(* Logix 5000 project; controller RG_Chopper vendor 1 type 14 code 235 rev 32.12; software revision 32.04; part 3 of 6 *)
(* tags used below, declared in another part *)
   _ILG101_GREEN_PB : BOOL;   // Green Light Pushbutton Local:1:O.Data.2
   ALARM_FATAL : BOOL;   // Fatal Alarm Stops All Operation
   ALARM_GATE_OPEN : BOOL;   // Gate Open
   ALARM_LIGHT_CUR : BOOL;   // Light Curtain Obstructed
   ALARM_NON_FATAL : BOOL;
   BLANK_LVL_DISP : BOOL;   // Disables Tank Level Display
   CIP_CAUSTIC_RUNNING : ALIAS FOR SIGNAL_OUT_RG_CHOPPER.4;
   CIP_CMPLT : BOOL;   // CIP Complete Indicator
   CIP_COMPLETE : ALIAS FOR SIGNAL_IN_RG_CHOPPER.4;
   CIP_CYC_ST : DINT;   // CIP Cycle Status HMI
   CIP_OUT : DINT;   // CIP Output Bits
   CIP_STEP : COUNTER;   // CIP Step Counter
   CIP_STEP_BIT : DINT;   // CIP Step Enable Bit
   CIP_STEP_DN : BOOL;   // CIP Step Done
   CIP_STEP_TMR : TIMER;   // CIP Step Timer
   CIP_STP_TM_TB : DINT[13];   // CIP Step Timer PreSet Table
   CIP_STRT_RUN : BOOL;   // CIP System Started
   CIP_WATER_RUNNING : ALIAS FOR SIGNAL_OUT_RG_CHOPPER.3;
   CYC_CIP : BOOL;   // CIP Cycle Running
   CYC_RUN : BOOL;   // Production Cycle Running
   CYC_ST : DINT;
   DBX101_AM : PUSH_PUSH_PB;   // DBX-101 Push-Push Button Control
   DBX101_AUX : BOOL;   // DBX-101 Agitator Motor Aux
   DBX101_CTL : HOA_CTRL_v2;   // DBX-101 Agitator Motor Control Block
   DBX101_CTL_ST : DINT;   // DBX-101 Control Status 0= Auto 1= Manual 2= Error
   DBX101_FAULT : BOOL;
   DBX101_MAN : PUSH_PUSH_PB;   // DBX-101 Manual Run Push-Push
   DBX101_MAN_RUN : BOOL;   // DBX-101 Manual Run
   DBX101_MAN_ST : DINT;   // DBX-101 Manual Control Status
   DBX101_PB : BOOL;   // DBX-101 Auto / Manual Push-Push Button
   DBX101_STS : DINT;   // DBX-101 Agitator Motor Status (HMI)
   DBX102_AM : PUSH_PUSH_PB;   // DBX-102 Push-Push Button Control
   DBX102_AUX : ALIAS FOR SIGNAL_IN_RG_CHOPPER.0;   // DBX-102 VFD Active AUX
   DBX102_CTL : HOA_CTRL_v2;   // DBX102 Product Discharge Pump Control Block
   DBX102_CTL_ST : DINT;   // DBX-102 Control Status 0= Auto 1= Manual 2= Error
   DBX102_M_FAULT : BOOL;   // DBX-102 Discharge Pump Drive or Motor Fault
   DBX102_MAN : PUSH_PUSH_PB;   // DBX-102 Manual Control Push-Push
   DBX102_MAN_RUN : BOOL;   // DBX-102 Manual Mode Run PB
   DBX102_MAN_ST : DINT;   // DBX-102 Manual Control Status
   DBX102_PB : BOOL;   // DBX-102 Auto / Manual Push-Push Button
   DBX102_SPD_AM : PUSH_PUSH_PB;   // DBX-102 Speed Push-Push Button Control
   DBX102_SPD_ST : DINT;   // DBX-102 VFD Speed Control Status 0= Auto 1= Manual 2= Error
   DBX102_STS : DINT;   // DBX-102 Product Pump Status (HMI)
   DBX102_VFD_FB : ANLG_SCALE;   // DBX-102 VFD Speed FB Scaling (HMI)
   DBX102_VFD_FB_SCL : REAL;   // DBX-102 Product Pump VFD Speed FB Scaling (HMI)
   DBX103_AM : PUSH_PUSH_PB;   // DBX-103 Push-Push Button Control
   DBX103_AUX : BOOL;   // DBX-103 Water Pump Aux
   DBX103_CTL : HOA_CTRL_v2;   // DBX-103 Hot Water Pump Control Block
   DBX103_CTL_ST : DINT;   // DBX-103 Control Status 1= Auto 2= Manual 3= Error
   DBX103_FAULT : BOOL;   // DBX-103 Hot Water Pump Fault
   DBX103_MAN : PUSH_PUSH_PB;   // DBX-103 Manual Run Push-Push
   DBX103_MAN_RUN : BOOL;   // DBX-101 Manual Run
   DBX103_MAN_ST : DINT;   // DBX-103 Manual Control Status
   DBX103_PB : BOOL;   // DBX-103 Auto / Manual Push-Push Button
   DBX103_STS : DINT;   // DBX-103 Hot Water Pump Status (HMI)
   DBX104_AM : PUSH_PUSH_PB;   // DBX-104 Push-Push Button Control
   DBX104_AUX : BOOL;   // DBX-104 VFD Active AUX
   DBX104_CTL : HOA_CTRL_v2;   // DBX-104 Reversing Motor Starter Control
   DBX104_CTL_ST : DINT;   // DBX-104 Control Status 0= Auto 1= Manual 2= Error
   DBX104_FAULT : BOOL;   // DBX-104 Dumper Elevator Drive Fault
   DBX104_M_FAULT : BOOL;   // DBX-104 Dumper Elevator Drive or Motor Fault
   DBX104_MAN : PUSH_PUSH_PB;   // DBX-104 Manual Control Push-Push
   DBX104_MAN_RUN : BOOL;   // DBX-104 Manual Mode Run PB
   DBX104_MAN_ST : DINT;   // DBX-104 Manual Control Status
   DBX104_PB : BOOL;   // DBX-104 Auto / Manual Push-Push Button
   DBX104_SPD_AM : PUSH_PUSH_PB;   // DBX-104 Speed Push-Push Button Control
   DBX104_SPD_ST : DINT;   // DBX-104 VFD Speed Control Status 0= Auto 1= Manual 2= Error
   DBX104_STS : DINT;   // DBX-104 Product Pump Status (HMI)
   DBX104_VFD_FB : ANLG_SCALE;   // DBX-104 VFD Speed FB Scaling (HMI)
   DBX104_VFD_FB_SCL : REAL;   // DBX-104 Product Pump VFD Speed FB Scaling (HMI)
   DL101_Scl : REAL;
   DTT102 : REAL;   // Discharge Product Temperature
   DWN_MKBK : BOOL;   // Elevator Down Make / Break LS_L1 Detection
   DWN_OT_AL : BOOL;   // New Dumper DOWN Over Travel Alarm
   Fault_ACK : BOOL;   // Fault Acknowledge
   Flash : BOOL;
   Gate_SW1 : DCI_MONITOR;   // Safety Switch Gate_SW1 SW105 A/B
   Gate_SW2 : DCI_MONITOR;   // Safety Switch Gate_SW2 SW108 A/B
   HI_PROD_TEMP_AL : BOOL;   // Product Temperature High Alarm
   HI_PROD_TEMP_SP : REAL;   // Product High Temperature Alarm SetPoint
   HI_TMP_TMR : TIMER;   // Product Temperature High Alarm Timer
   HMI_USER : STRING;   // Current Logged HMI User
   ILG104_GREEN_STACK : BOOL;   // Stack Light Green
   ILG105_YELLOW_STACK : BOOL;   // Stack Light Yellow
   ILG106_RED_STACK : BOOL;   // Stack Light Red
   L_CRASH_ALM : BOOL;   // New Dumper Lower CRASH Alarm
   LSS_LOT1 : BOOL;   // New Dumper LOWER OVER TRAVEL Limit Switch
   LVL_BLANK_SP : REAL;   // Real Value Below Blanks Level Display
   LVL_LO_TMR : TIMER;   // Low Tank Level Alarm Debounce Timer
   M104S_DWN_CTL : CONFIGURABLE_ROUT;   // DBX-104 Dump Elevator Safety Starter Down Output
   M104S_STRT_CTL : CONFIGURABLE_ROUT;   // DBX-104 Dump Elevator Safety Starter Enable Output
   M104S_UP_CTL : CONFIGURABLE_ROUT;   // DBX-104 Dump Elevator Safety Starter UP Output
   NO_USER : BOOL;   // No HMI User Logged on
   ONESHOT : DINT;   // One-shot Word
   PROC_TMR : TIMER[16];   // Process Timers
   S_ESTOP : BOOL;   // Safety ESTOP
   SHTDWN_ACTV : BOOL;   // System Shutdown is In Progress
   SHTDWN_CMPLT : BOOL;   // System Shutdown Complete
   SHUTDOWN : DINT;   // System Shutdown Control Bits
   SIGNAL_OUT_RG_CHOPPER : DINT;
   START_CMPLT : BOOL;   // System Start up Complete
   SW102_STOP_PB : BOOL;   // Stop PB HMI
   SW103_CIP_PB : BOOL;   // CIP PB HMI
   SW104_ESTOP : BOOL;   // Safety E-Stop SW-104
   SW106_LC : LIGHT_CURTAIN;   // Safety SW106 Light Curain
   SW107_TANK_LID : BOOL;   // Tank Lid Safety Switch Active
   SYS_OK : BOOL;   // System OK No Fatal Alarms
   SYS_STRT_RUN : BOOL;   // System Start / Run
   TCV101_CTL : PID;   // PCV-101 PID Temperature Control
   UP_MKBK : BOOL;   // Elevator Down Make / Break LS_U1 Detection
   UP_OT_AL : BOOL;   // New Dumper UP Over Travel Alarm
   USER_ON : BOOL;   // There IS a valid HMI User Logged On
   WTR_HI_TEMP : BOOL;   // High Water Temperature Alarm
   WTR_HI_TMR : TIMER;   // High Water Temperature Alarm Debounce Timer

PROGRAM MainProgram   (* main routine MainRoutine *)
VAR
   L2_FAIL_TMR : TIMER := (PRE := 4000);   // LSSL2 Fail Always Open Detect
   LSSL2_FAIL : BOOL;   // Lower Safety Limit Switch LSS-L2 Fail
   LSSL2_FAIL2 : BOOL;   // Lower Safety Limit Switch LSS-L2 Mode 2
   LSSU2_FAIL : BOOL;   // Upper Safety Limit Switch LSS-U2 Fail
   LSSU2_FAIL2 : BOOL;   // Upper Safety Limit Switch USS-L2 Mode 2
   U2_FAIL_TMR : TIMER := (PRE := 4000);   // LSSU2 Fail Always Open Detect
END_VAR

ROUTINE ALARMS   (* ladder *)
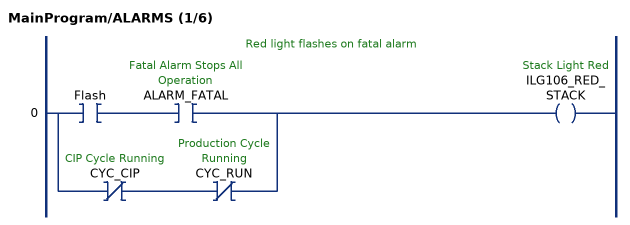
   // Red light flashes on fatal alarm
   0: [XIC(Flash) XIC(ALARM_FATAL) ,XIO(CYC_CIP) XIO(CYC_RUN) ]OTE(ILG106_RED_STACK);
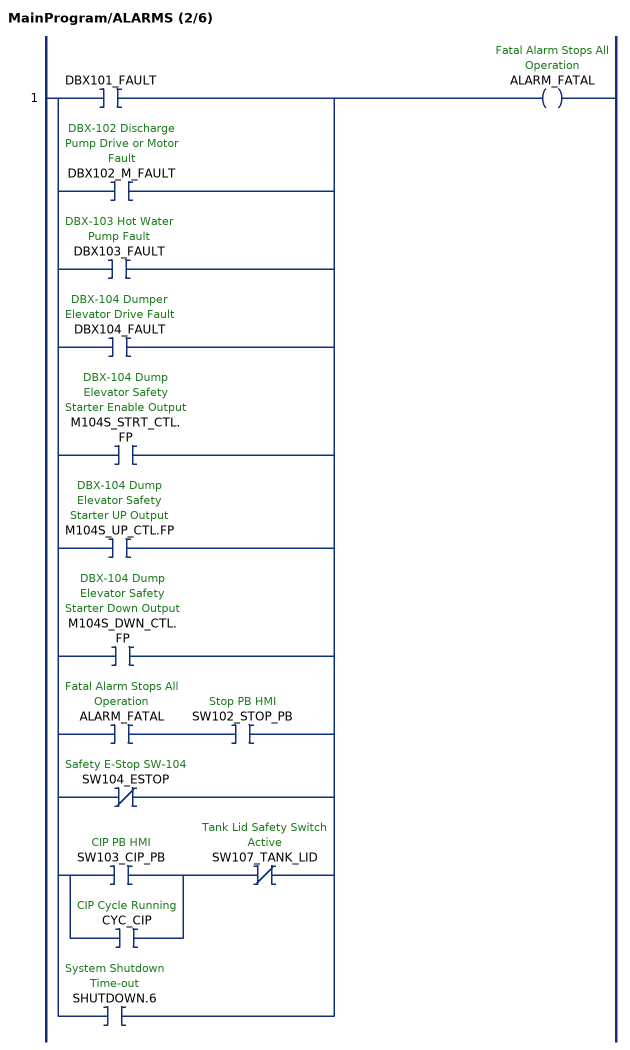
   1: [XIC(DBX101_FAULT) ,XIC(DBX102_M_FAULT) ,XIC(DBX103_FAULT) ,XIC(DBX104_FAULT) ,XIC(M104S_STRT_CTL.FP) ,XIC(M104S_UP_CTL.FP) ,XIC(M104S_DWN_CTL.FP) ,XIC(ALARM_FATAL) XIC(SW102_STOP_PB) ,XIO(SW104_ESTOP) ,[XIC(SW103_CIP_PB) ,XIC(CYC_CIP) ] XIO(SW107_TANK_LID) ,XIC(SHUTDOWN.6) ]OTE(ALARM_FATAL);
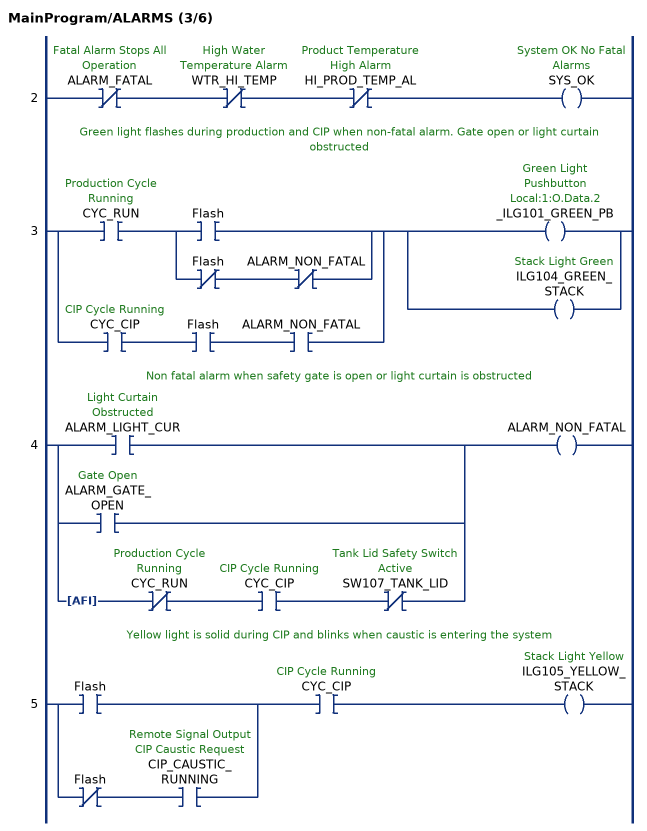
   2: XIO(ALARM_FATAL)XIO(WTR_HI_TEMP)XIO(HI_PROD_TEMP_AL)OTE(SYS_OK);
   // Green light flashes during production and CIP when non-fatal alarm. Gate open or light curtain obstructed
   3: [XIC(CYC_RUN) [XIC(Flash) ,XIO(Flash) XIO(ALARM_NON_FATAL) ] ,XIC(CYC_CIP) XIC(Flash) XIC(ALARM_NON_FATAL) ][OTE(_ILG101_GREEN_PB) ,OTE(ILG104_GREEN_STACK) ];
   // Non fatal alarm when safety gate is open or light curtain is obstructed
   4: [XIC(ALARM_LIGHT_CUR) ,XIC(ALARM_GATE_OPEN) ,AFI() XIO(CYC_RUN) XIC(CYC_CIP) XIO(SW107_TANK_LID) ]OTE(ALARM_NON_FATAL);
   // Yellow light is solid during CIP and blinks when caustic is entering the system
   5: [XIC(Flash) ,XIO(Flash) XIC(CIP_CAUSTIC_RUNNING) ]XIC(CYC_CIP)OTE(ILG105_YELLOW_STACK);
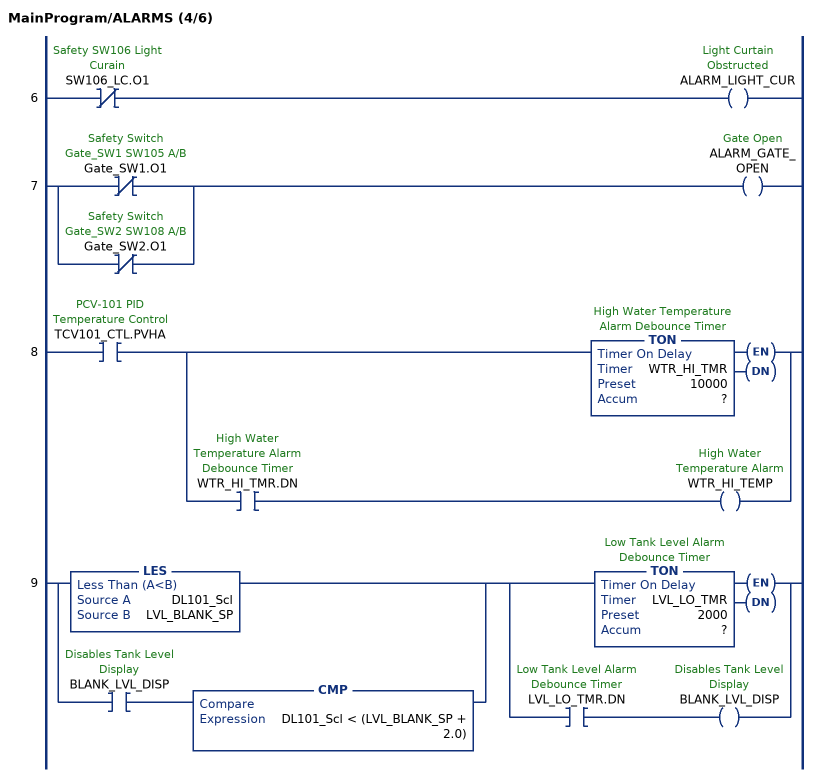
   6: XIO(SW106_LC.O1)OTE(ALARM_LIGHT_CUR);
   7: [XIO(Gate_SW1.O1) ,XIO(Gate_SW2.O1) ]OTE(ALARM_GATE_OPEN);
   8: XIC(TCV101_CTL.PVHA)[TON(WTR_HI_TMR,?,?) ,XIC(WTR_HI_TMR.DN) OTE(WTR_HI_TEMP) ];
   9: [LES(DL101_Scl,LVL_BLANK_SP) ,XIC(BLANK_LVL_DISP) CMP(DL101_Scl < (LVL_BLANK_SP + 2.0)) ][TON(LVL_LO_TMR,?,?) ,XIC(LVL_LO_TMR.DN) OTE(BLANK_LVL_DISP) ];
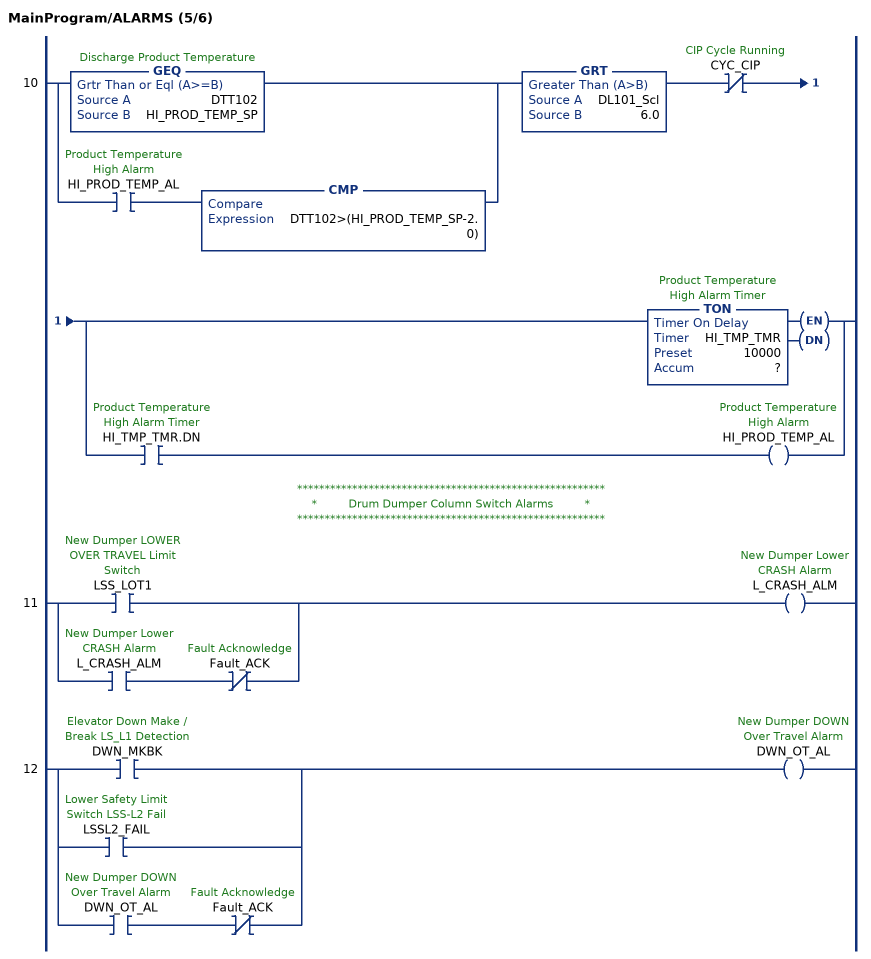
   10: [GEQ(DTT102,HI_PROD_TEMP_SP) ,XIC(HI_PROD_TEMP_AL) CMP(DTT102>(HI_PROD_TEMP_SP-2.0)) ]GRT(DL101_Scl,6.0)XIO(CYC_CIP)[TON(HI_TMP_TMR,?,?) ,XIC(HI_TMP_TMR.DN) OTE(HI_PROD_TEMP_AL) ];
   // ********************************************************
   // *         Drum Dumper Column Switch Alarms         *
   // ********************************************************
   11: [XIC(LSS_LOT1) ,XIC(L_CRASH_ALM) XIO(Fault_ACK) ]OTE(L_CRASH_ALM);
   12: [XIC(DWN_MKBK) ,XIC(LSSL2_FAIL) ,XIC(DWN_OT_AL) XIO(Fault_ACK) ]OTE(DWN_OT_AL);
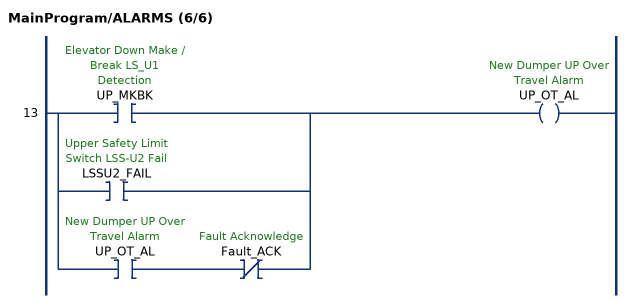
   13: [XIC(UP_MKBK) ,XIC(LSSU2_FAIL) ,XIC(UP_OT_AL) XIO(Fault_ACK) ]OTE(UP_OT_AL);
END_ROUTINE

ROUTINE CIP   (* ladder *)
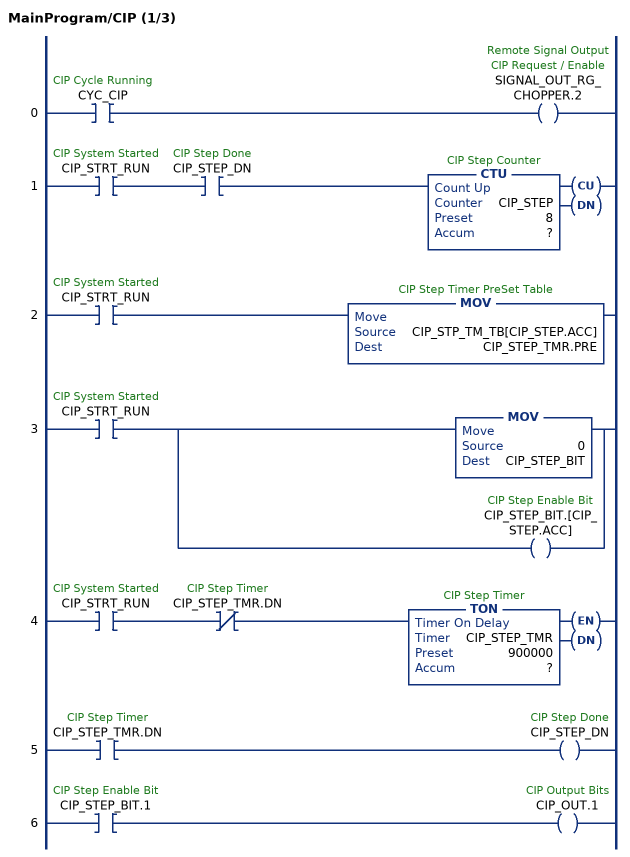
   0: XIC(CYC_CIP)OTE(SIGNAL_OUT_RG_CHOPPER.2);
   1: XIC(CIP_STRT_RUN)XIC(CIP_STEP_DN)CTU(CIP_STEP,?,?);
   2: XIC(CIP_STRT_RUN)MOV(CIP_STP_TM_TB[CIP_STEP.ACC],CIP_STEP_TMR.PRE);
   3: XIC(CIP_STRT_RUN)[MOV(0,CIP_STEP_BIT) ,OTE(CIP_STEP_BIT.[CIP_STEP.ACC]) ];
   4: XIC(CIP_STRT_RUN)XIO(CIP_STEP_TMR.DN)TON(CIP_STEP_TMR,?,?);
   5: XIC(CIP_STEP_TMR.DN)OTE(CIP_STEP_DN);
   6: XIC(CIP_STEP_BIT.1)OTE(CIP_OUT.1);
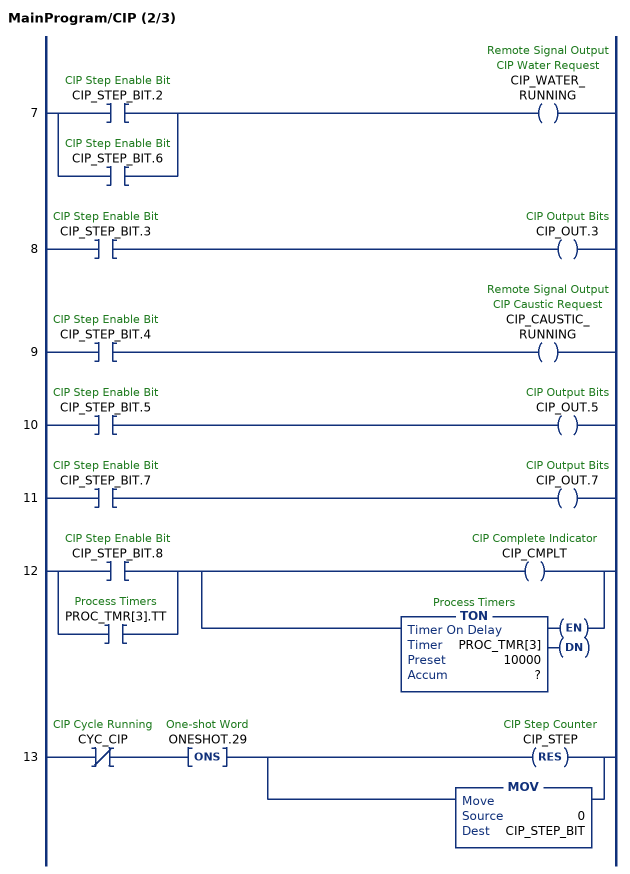
   7: [XIC(CIP_STEP_BIT.2) ,XIC(CIP_STEP_BIT.6) ]OTE(CIP_WATER_RUNNING);
   8: XIC(CIP_STEP_BIT.3)OTE(CIP_OUT.3);
   9: XIC(CIP_STEP_BIT.4)OTE(CIP_CAUSTIC_RUNNING);
   10: XIC(CIP_STEP_BIT.5)OTE(CIP_OUT.5);
   11: XIC(CIP_STEP_BIT.7)OTE(CIP_OUT.7);
   12: [XIC(CIP_STEP_BIT.8) ,XIC(PROC_TMR[3].TT) ][OTE(CIP_CMPLT) ,TON(PROC_TMR[3],?,?) ];
   13: XIO(CYC_CIP)ONS(ONESHOT.29)[RES(CIP_STEP) ,MOV(0,CIP_STEP_BIT) ];
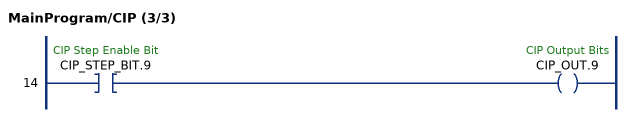
   14: XIC(CIP_STEP_BIT.9)OTE(CIP_OUT.9);
END_ROUTINE

ROUTINE HMI   (* ladder *)
// HMI Interface Code
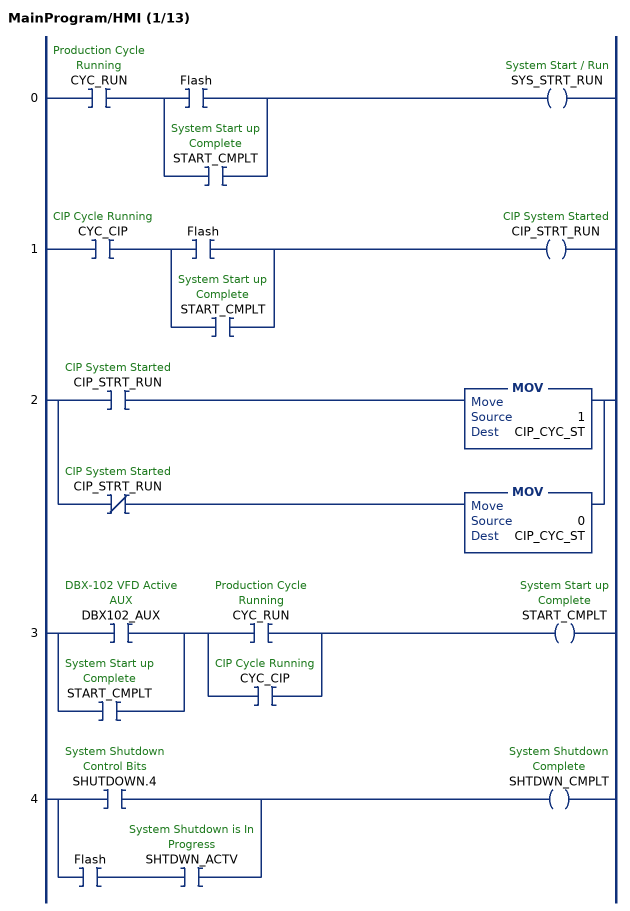
   0: XIC(CYC_RUN)[XIC(Flash) ,XIC(START_CMPLT) ]OTE(SYS_STRT_RUN);
   1: XIC(CYC_CIP)[XIC(Flash) ,XIC(START_CMPLT) ]OTE(CIP_STRT_RUN);
   2: [XIC(CIP_STRT_RUN) MOV(1,CIP_CYC_ST) ,XIO(CIP_STRT_RUN) MOV(0,CIP_CYC_ST) ];
   3: [XIC(DBX102_AUX) ,XIC(START_CMPLT) ][XIC(CYC_RUN) ,XIC(CYC_CIP) ]OTE(START_CMPLT);
   4: [XIC(SHUTDOWN.4) ,XIC(Flash) XIC(SHTDWN_ACTV) ]OTE(SHTDWN_CMPLT);
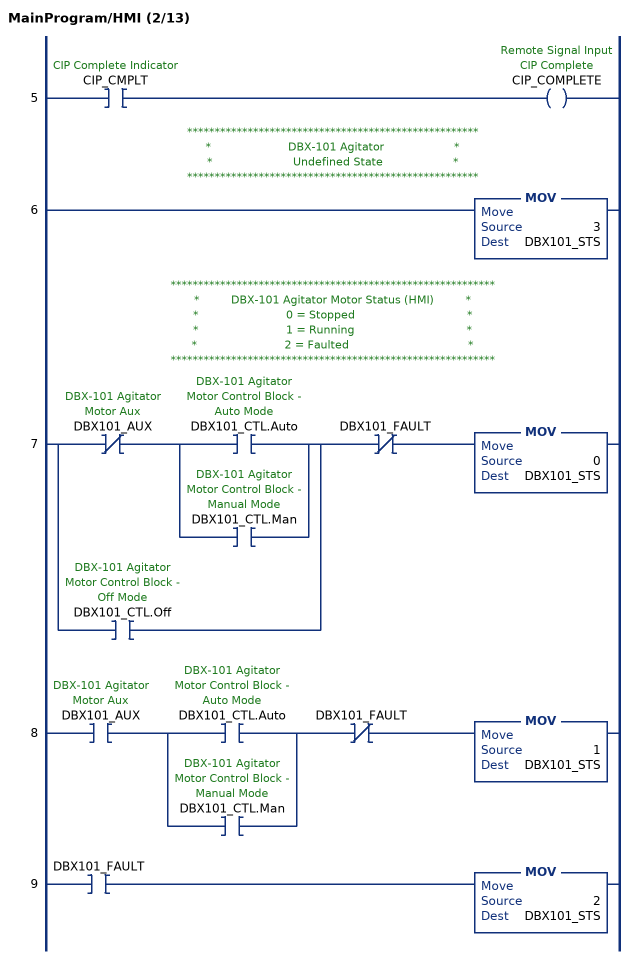
   5: XIC(CIP_CMPLT)OTE(CIP_COMPLETE);
   // *****************************************************
   // *                      DBX-101 Agitator                    *
   // *                       Undefined State                    *
   // *****************************************************
   6: MOV(3,DBX101_STS);
   // ***********************************************************
   // *         DBX-101 Agitator Motor Status (HMI)         *
   // *                         0 = Stopped                                *
   // *                         1 = Running                                *
   // *                         2 = Faulted                                  *
   // ***********************************************************
   7: [XIO(DBX101_AUX) [XIC(DBX101_CTL.Auto) ,XIC(DBX101_CTL.Man) ] ,XIC(DBX101_CTL.Off) ]XIO(DBX101_FAULT)MOV(0,DBX101_STS);
   8: XIC(DBX101_AUX)[XIC(DBX101_CTL.Auto) ,XIC(DBX101_CTL.Man) ]XIO(DBX101_FAULT)MOV(1,DBX101_STS);
   9: XIC(DBX101_FAULT)MOV(2,DBX101_STS);
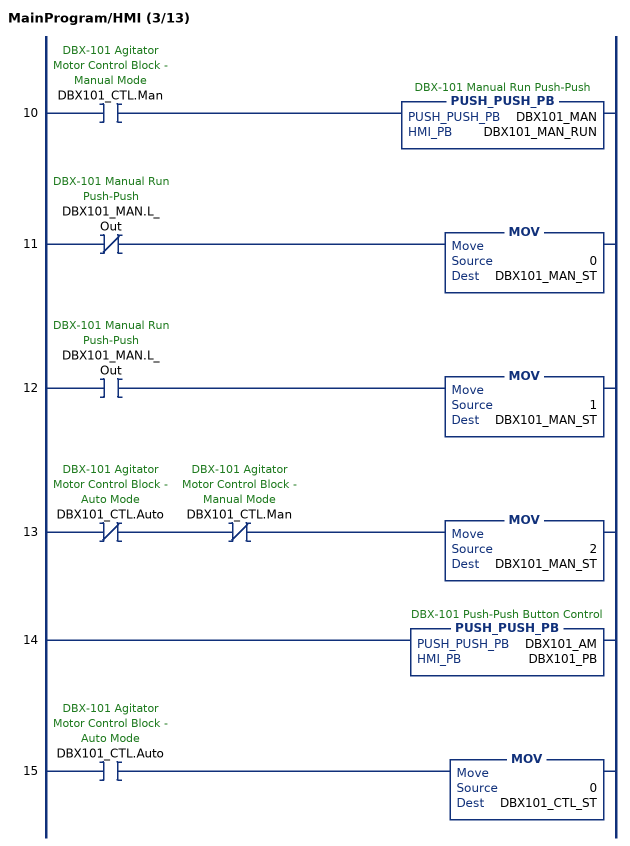
   10: XIC(DBX101_CTL.Man)PUSH_PUSH_PB(DBX101_MAN,DBX101_MAN_RUN);
   11: XIO(DBX101_MAN.L_Out)MOV(0,DBX101_MAN_ST);
   12: XIC(DBX101_MAN.L_Out)MOV(1,DBX101_MAN_ST);
   13: XIO(DBX101_CTL.Auto)XIO(DBX101_CTL.Man)MOV(2,DBX101_MAN_ST);
   14: PUSH_PUSH_PB(DBX101_AM,DBX101_PB);
   15: XIC(DBX101_CTL.Auto)MOV(0,DBX101_CTL_ST);
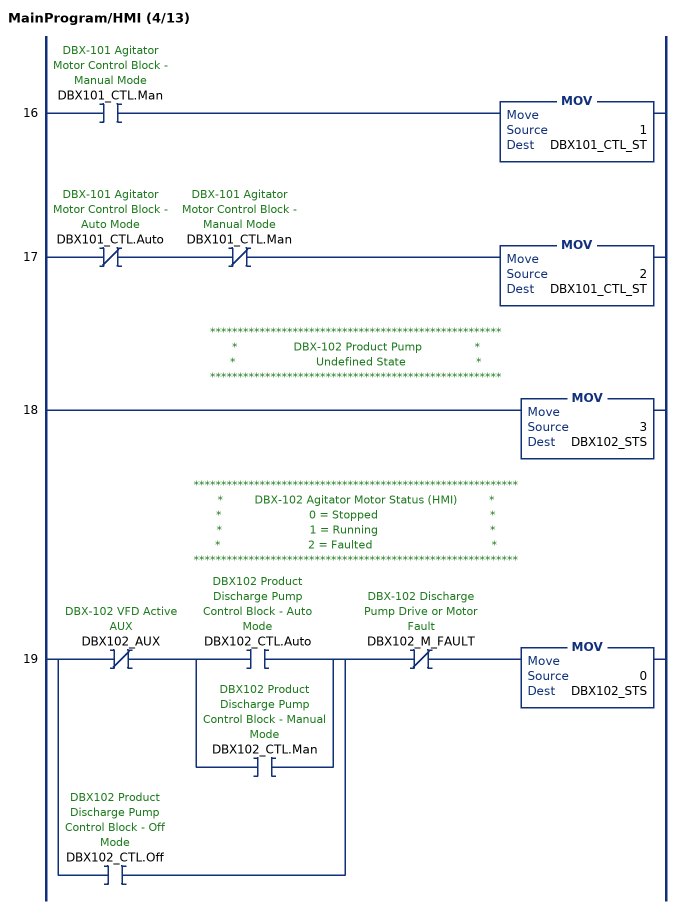
   16: XIC(DBX101_CTL.Man)MOV(1,DBX101_CTL_ST);
   17: XIO(DBX101_CTL.Auto)XIO(DBX101_CTL.Man)MOV(2,DBX101_CTL_ST);
   // *****************************************************
   // *                DBX-102 Product Pump               *
   // *                       Undefined State                    *
   // *****************************************************
   18: MOV(3,DBX102_STS);
   // ***********************************************************
   // *         DBX-102 Agitator Motor Status (HMI)         *
   // *                         0 = Stopped                                *
   // *                         1 = Running                                *
   // *                         2 = Faulted                                  *
   // ***********************************************************
   19: [XIO(DBX102_AUX) [XIC(DBX102_CTL.Auto) ,XIC(DBX102_CTL.Man) ] ,XIC(DBX102_CTL.Off) ]XIO(DBX102_M_FAULT)MOV(0,DBX102_STS);
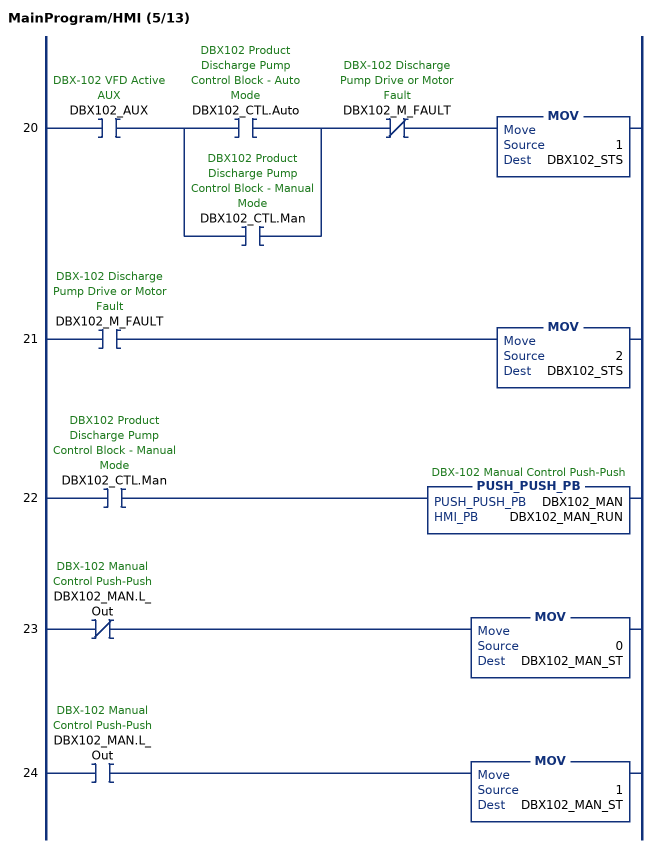
   20: XIC(DBX102_AUX)[XIC(DBX102_CTL.Auto) ,XIC(DBX102_CTL.Man) ]XIO(DBX102_M_FAULT)MOV(1,DBX102_STS);
   21: XIC(DBX102_M_FAULT)MOV(2,DBX102_STS);
   22: XIC(DBX102_CTL.Man)PUSH_PUSH_PB(DBX102_MAN,DBX102_MAN_RUN);
   23: XIO(DBX102_MAN.L_Out)MOV(0,DBX102_MAN_ST);
   24: XIC(DBX102_MAN.L_Out)MOV(1,DBX102_MAN_ST);
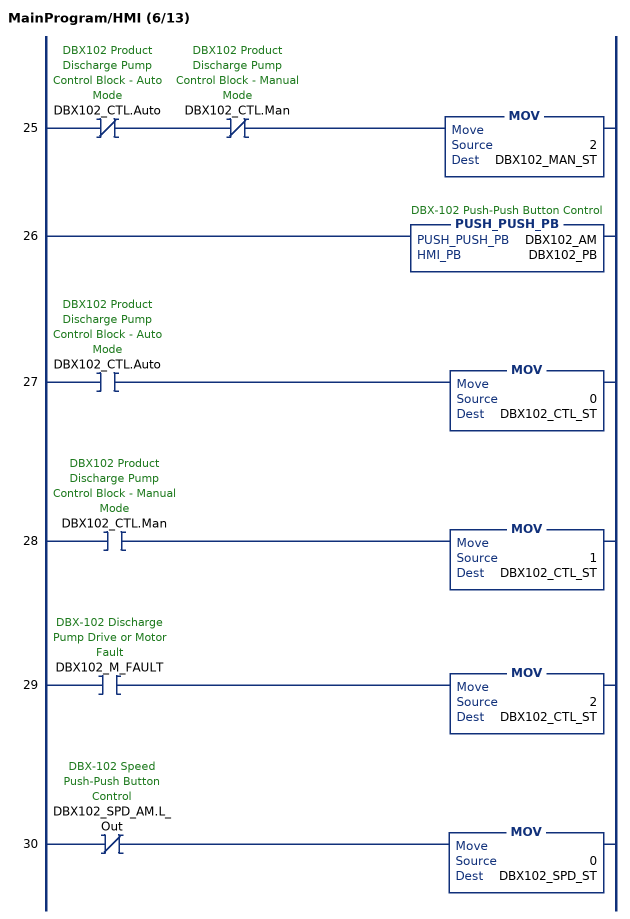
   25: XIO(DBX102_CTL.Auto)XIO(DBX102_CTL.Man)MOV(2,DBX102_MAN_ST);
   26: PUSH_PUSH_PB(DBX102_AM,DBX102_PB);
   27: XIC(DBX102_CTL.Auto)MOV(0,DBX102_CTL_ST);
   28: XIC(DBX102_CTL.Man)MOV(1,DBX102_CTL_ST);
   29: XIC(DBX102_M_FAULT)MOV(2,DBX102_CTL_ST);
   30: XIO(DBX102_SPD_AM.L_Out)MOV(0,DBX102_SPD_ST);
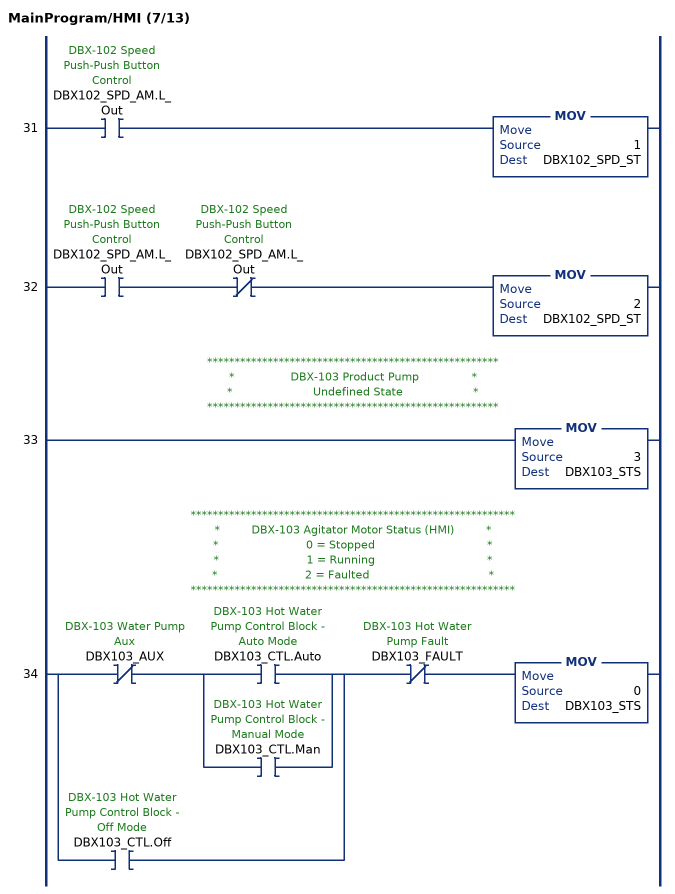
   31: XIC(DBX102_SPD_AM.L_Out)MOV(1,DBX102_SPD_ST);
   32: XIC(DBX102_SPD_AM.L_Out)XIO(DBX102_SPD_AM.L_Out)MOV(2,DBX102_SPD_ST);
   // *****************************************************
   // *                DBX-103 Product Pump               *
   // *                       Undefined State                    *
   // *****************************************************
   33: MOV(3,DBX103_STS);
   // ***********************************************************
   // *         DBX-103 Agitator Motor Status (HMI)         *
   // *                         0 = Stopped                                *
   // *                         1 = Running                                *
   // *                         2 = Faulted                                  *
   // ***********************************************************
   34: [XIO(DBX103_AUX) [XIC(DBX103_CTL.Auto) ,XIC(DBX103_CTL.Man) ] ,XIC(DBX103_CTL.Off) ]XIO(DBX103_FAULT)MOV(0,DBX103_STS);
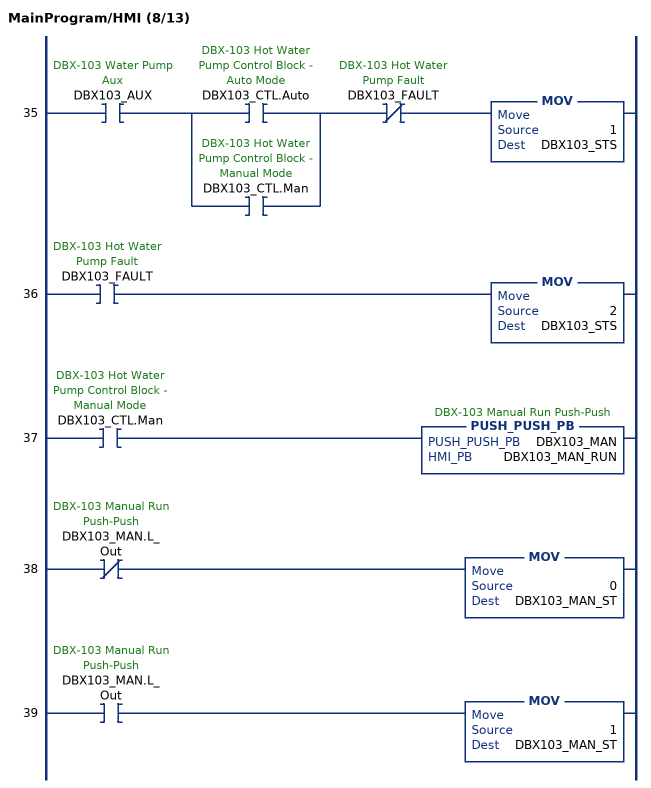
   35: XIC(DBX103_AUX)[XIC(DBX103_CTL.Auto) ,XIC(DBX103_CTL.Man) ]XIO(DBX103_FAULT)MOV(1,DBX103_STS);
   36: XIC(DBX103_FAULT)MOV(2,DBX103_STS);
   37: XIC(DBX103_CTL.Man)PUSH_PUSH_PB(DBX103_MAN,DBX103_MAN_RUN);
   38: XIO(DBX103_MAN.L_Out)MOV(0,DBX103_MAN_ST);
   39: XIC(DBX103_MAN.L_Out)MOV(1,DBX103_MAN_ST);
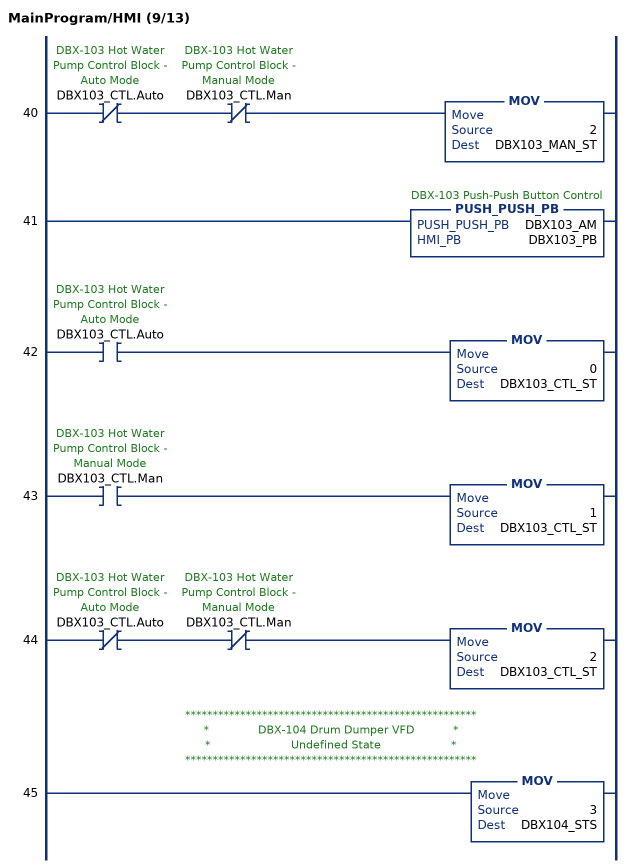
   40: XIO(DBX103_CTL.Auto)XIO(DBX103_CTL.Man)MOV(2,DBX103_MAN_ST);
   41: PUSH_PUSH_PB(DBX103_AM,DBX103_PB);
   42: XIC(DBX103_CTL.Auto)MOV(0,DBX103_CTL_ST);
   43: XIC(DBX103_CTL.Man)MOV(1,DBX103_CTL_ST);
   44: XIO(DBX103_CTL.Auto)XIO(DBX103_CTL.Man)MOV(2,DBX103_CTL_ST);
   // *****************************************************
   // *              DBX-104 Drum Dumper VFD           *
   // *                       Undefined State                    *
   // *****************************************************
   45: MOV(3,DBX104_STS);
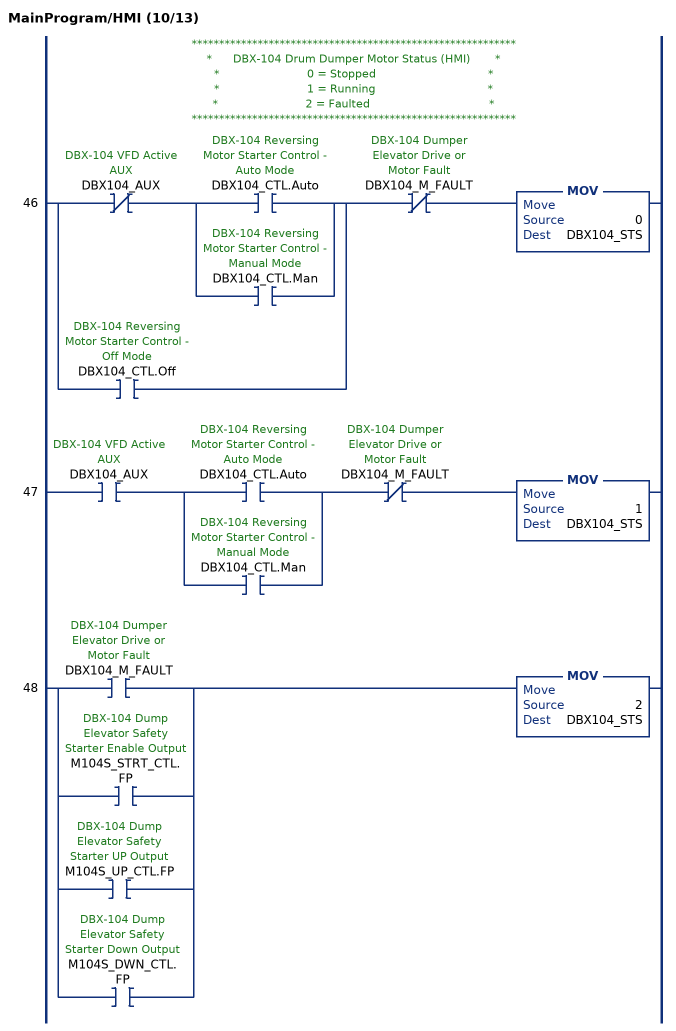
   // ***********************************************************
   // *      DBX-104 Drum Dumper Motor Status (HMI)       *
   // *                         0 = Stopped                                *
   // *                         1 = Running                                *
   // *                         2 = Faulted                                  *
   // ***********************************************************
   46: [XIO(DBX104_AUX) [XIC(DBX104_CTL.Auto) ,XIC(DBX104_CTL.Man) ] ,XIC(DBX104_CTL.Off) ]XIO(DBX104_M_FAULT)MOV(0,DBX104_STS);
   47: XIC(DBX104_AUX)[XIC(DBX104_CTL.Auto) ,XIC(DBX104_CTL.Man) ]XIO(DBX104_M_FAULT)MOV(1,DBX104_STS);
   48: [XIC(DBX104_M_FAULT) ,XIC(M104S_STRT_CTL.FP) ,XIC(M104S_UP_CTL.FP) ,XIC(M104S_DWN_CTL.FP) ]MOV(2,DBX104_STS);
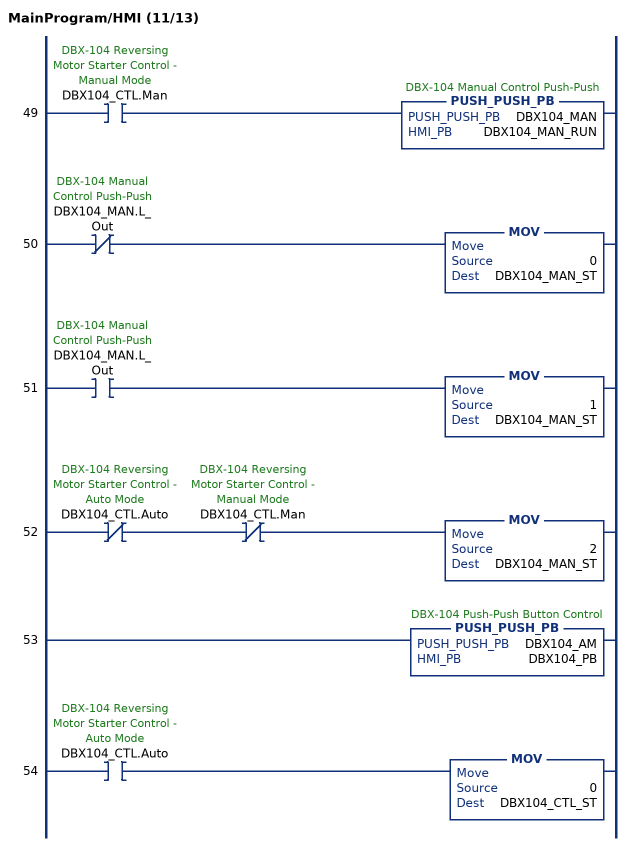
   49: XIC(DBX104_CTL.Man)PUSH_PUSH_PB(DBX104_MAN,DBX104_MAN_RUN);
   50: XIO(DBX104_MAN.L_Out)MOV(0,DBX104_MAN_ST);
   51: XIC(DBX104_MAN.L_Out)MOV(1,DBX104_MAN_ST);
   52: XIO(DBX104_CTL.Auto)XIO(DBX104_CTL.Man)MOV(2,DBX104_MAN_ST);
   53: PUSH_PUSH_PB(DBX104_AM,DBX104_PB);
   54: XIC(DBX104_CTL.Auto)MOV(0,DBX104_CTL_ST);
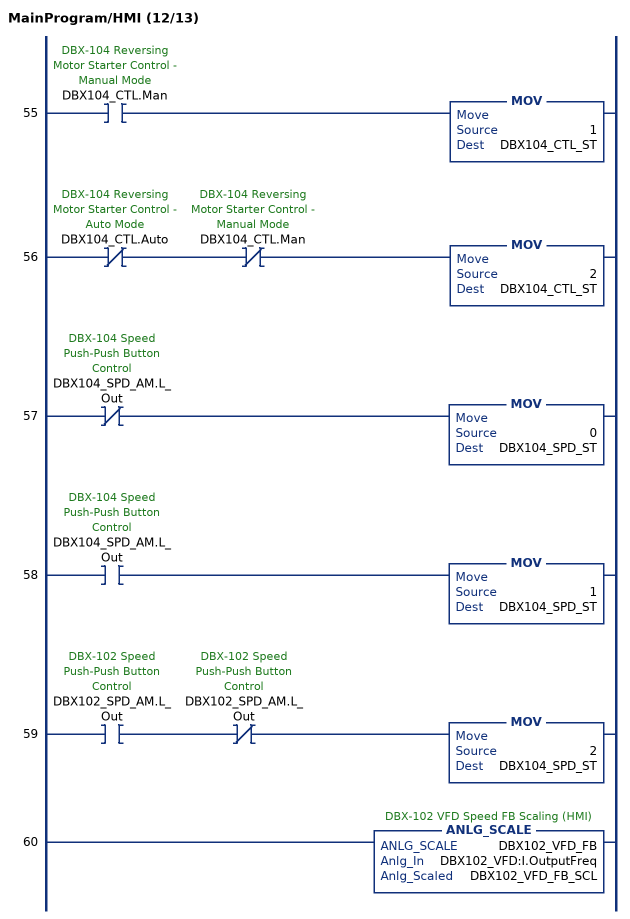
   55: XIC(DBX104_CTL.Man)MOV(1,DBX104_CTL_ST);
   56: XIO(DBX104_CTL.Auto)XIO(DBX104_CTL.Man)MOV(2,DBX104_CTL_ST);
   57: XIO(DBX104_SPD_AM.L_Out)MOV(0,DBX104_SPD_ST);
   58: XIC(DBX104_SPD_AM.L_Out)MOV(1,DBX104_SPD_ST);
   59: XIC(DBX102_SPD_AM.L_Out)XIO(DBX102_SPD_AM.L_Out)MOV(2,DBX104_SPD_ST);
   60: ANLG_SCALE(DBX102_VFD_FB,DBX102_VFD:I.OutputFreq,DBX102_VFD_FB_SCL);
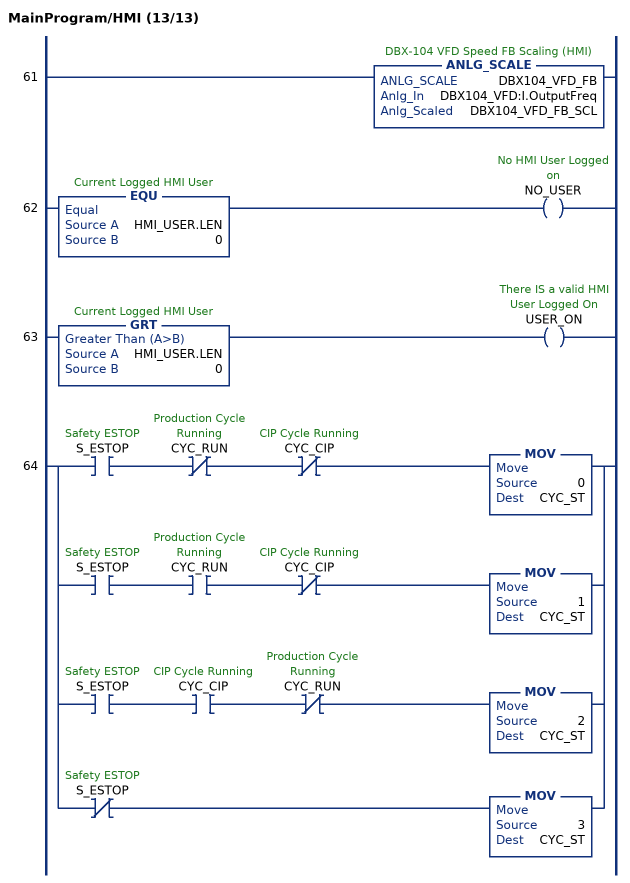
   61: ANLG_SCALE(DBX104_VFD_FB,DBX104_VFD:I.OutputFreq,DBX104_VFD_FB_SCL);
   62: EQU(HMI_USER.LEN,0)OTE(NO_USER);
   63: GRT(HMI_USER.LEN,0)OTE(USER_ON);
   64: [XIC(S_ESTOP) XIO(CYC_RUN) XIO(CYC_CIP) MOV(0,CYC_ST) ,XIC(S_ESTOP) XIC(CYC_RUN) XIO(CYC_CIP) MOV(1,CYC_ST) ,XIC(S_ESTOP) XIC(CYC_CIP) XIO(CYC_RUN) MOV(2,CYC_ST) ,XIO(S_ESTOP) MOV(3,CYC_ST) ];
END_ROUTINE
